PROGRAM FAST
VAR
END_VAR

END_PROGRAM

(* stored: Version 1.1.0.1, ProductVersion 3.1.4022.18
   POU FAST: Id {346f77cf-e7e3-4cc8-8cea-585644fa2845}, SpecialFunc None *)
